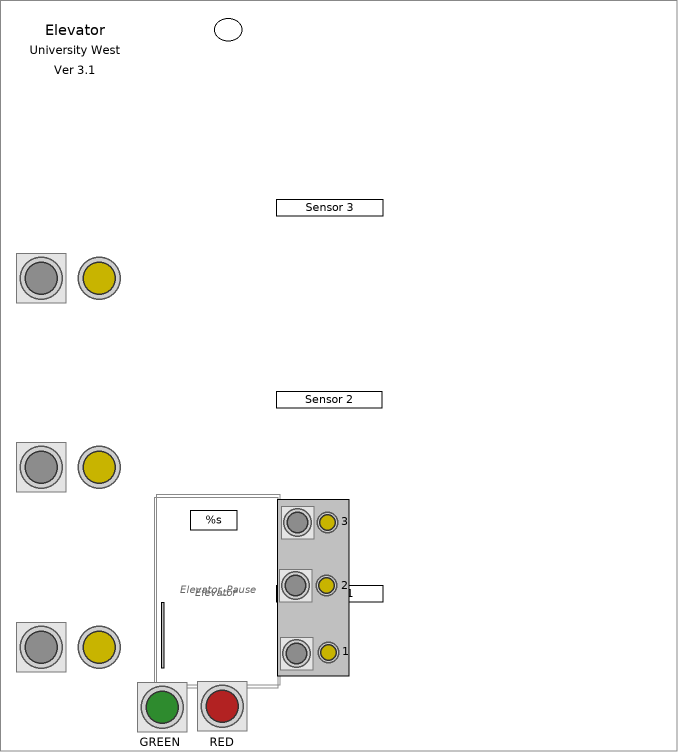
VISUALIZATION ElevatorSimulator  // 678x752
    Frame (154,497 124x191)
        shows Elevator()
        pReferences[0]: m_Input_RUNNING=Global_Variables.libMotorRunning, m_Input_LIMIT=Global_Variables.libTopLimit
        p2738717112: -Process.iElevatPos
    Frame (156,494 124x191), invisible if: true
        shows Elevator_Pause()
        p2738717112: -Process.iElevatPos
    Rectangle (30,340 100x80), "DANGER! Door not closed!"
    Rectangle (21,332 120x100), invisible if: Process.xWarning
    Rectangle (276,585 107x17), "Sensor 1", colour toggle: GVL.qxElevatLevel1
    Rectangle (276,391 106x17), "Sensor 2", colour toggle: GVL.qxElevatLevel2
    Rectangle (276,199 107x17), "Sensor 3", colour toggle: GVL.qxElevatLevel3
    Polyline (74,489)
    Polyline (266,5)
    Polyline (74,299)
    Polyline (74,109)
    Polyline (74,668)
    Polyline (142,6)
    Polyline (143,108)
    Ellipse (214,18 28x23), colour toggle: Process.xMotorRunning
    Rectangle (20,40 110x20), "University West"
    Rectangle (20,60 110x20), "Ver 3.1"
    Rectangle (161,602 3x66)
        p2738717112: -Process.iElevatPos
        p874137650: Process.iDoorPosition*2
    Rectangle (20,20 110x20), "Elevator"
    Lamp1 (74,622 50x50), variable: GVL.ixLampLevel1, style: Lamp-Lamp1-Yellow
    PushSwitch (16,622 50x50), variable: GVL.qxButtLevel1, behaviour: TAP, style: Switch-PushSwitch-Gray
    Lamp1 (74,442 50x50), variable: GVL.ixLampLevel2, style: Lamp-Lamp1-Yellow
    PushSwitch (16,442 50x50), variable: GVL.qxButtLevel2, behaviour: TAP, style: Switch-PushSwitch-Gray
    Lamp1 (74,253 50x50), variable: GVL.ixLampLevel3, style: Lamp-Lamp1-Yellow
    PushSwitch (16,253 50x50), variable: GVL.qxButtLevel3, behaviour: TAP, style: Switch-PushSwitch-Gray
    PushSwitch (137,682 50x50), variable: GVL.qxButtGreen, behaviour: TAP, style: Switch-PushSwitch-Green
    PushSwitch (197,681 50x50), variable: Process.xButtRedInv, behaviour: TAP, style: Switch-PushSwitch-Red
    Line (677,73)
    Group (277,499 79x177)
        p2738717112: -Process.iElevatPos
        Rectangle (0,0 72x177)
        Lamp1 (39,141 25x25), variable: GVL.ixLampElevat1, style: Lamp-Lamp1-Yellow
        Lamp1 (37,74 25x25), variable: GVL.ixLampElevat2, style: Lamp-Lamp1-Yellow
        Lamp1 (38,11 25x25), variable: GVL.ixLampElevat3, style: Lamp-Lamp1-Yellow
        Label (57,9 21x27), "3"
        Label (58,139 21x27), "1"
        Label (57,73 21x27), "2"
        PushSwitch (3,137 33x35), variable: GVL.qxButtElevat1, behaviour: TAP, style: Switch-PushSwitch-Gray
        PushSwitch (2,69 33x35), variable: GVL.qxButtElevat2, behaviour: TAP, style: Switch-PushSwitch-Gray
        PushSwitch (4,6 33x35), variable: GVL.qxButtElevat3, behaviour: TAP, style: Switch-PushSwitch-Gray
    Rectangle (190,510 47x20), "%s", text variable: GVL.iiDisplayElevat
        p2738717112: -Process.iElevatPos
    Rectangle (124,732 72x20), "GREEN"
    Rectangle (186,732 72x20), "RED"
END_VISUALIZATION

(* stored: Version 1.1.0.1
   Visu ElevatorSimulator: Id {a9b597a5-fe73-4c17-b3ee-267c0b4cfd36} *)
